// TIA Portal V20 export
DATA_BLOCK "DB_Manual"   // DB4
{ S7_Optimized_Access := 'TRUE' }
// stored: MemoryReserve 100
   VAR
      Modo_Activo : Bool;
      HMI_C1_Sale : Bool;
      HMI_C1_Entra : Bool;
      HMI_C2_Sale : Bool;
      HMI_C2_Entra : Bool;
      "HMI_M_90°" : Bool;
      "HMI_M_0°" : Bool;
   END_VAR
BEGIN
END_DATA_BLOCK
